(* IEC 61131-3 sources: RL_MAR/experiments/comparison/autoplc/results/gpt-4o-mini_20260511_164212/med_70, 1 file *)

(* ---- med_70_1.st ---- *)
FUNCTION_BLOCK EggIncubatorControl
    VAR_INPUT
        StartButton : BOOL; (* Input for starting the incubation process *)
        StopButton : BOOL; (* Input for stopping the incubation process *)
        TemperatureSensor : REAL; (* Input for temperature reading in °C *)
        HumiditySensor : REAL; (* Input for humidity reading in % *)
    END_VAR

    VAR_OUTPUT
        HeatingElement : BOOL; (* Output for controlling the heating element *)
        Humidifier : BOOL; (* Output for controlling the humidifier *)
        EggTurningMotor : BOOL; (* Output for controlling the egg turning motor *)
        IncubationInProgress : BOOL; (* Indicator for an ongoing incubation process *)
    END_VAR

    VAR
        TargetTemperature : REAL; (* Target temperature in °C *)
        TargetHumidity : REAL; (* Target humidity in % *)
        TurnIntervalSeconds : INT; (* Interval for turning eggs (1 hour in seconds) *)
        TurnTimerSeconds : INT; (* Timer for egg turning cycle in seconds *)
    END_VAR

    // Initialize control parameters
    TargetTemperature := 37.5;
    TargetHumidity := 50.0;
    TurnIntervalSeconds := 3600;
    TurnTimerSeconds := 0;

    // Main control logic
    IF StartButton AND NOT IncubationInProgress THEN
        IncubationInProgress := TRUE; // Start incubation
    END_IF;

    IF StopButton THEN
        IncubationInProgress := FALSE; // Stop incubation
        HeatingElement := FALSE; // Turn off heating element
        Humidifier := FALSE; // Turn off humidifier
        EggTurningMotor := FALSE; // Turn off egg turning motor
        TurnTimerSeconds := 0; // Reset timer
    END_IF;

    // Temperature control logic
    IF TemperatureSensor < TargetTemperature THEN
        HeatingElement := TRUE; // Turn on heating element
    ELSE
        HeatingElement := FALSE; // Turn off heating element
    END_IF;

    // Humidity control logic
    IF HumiditySensor < TargetHumidity THEN
        Humidifier := TRUE; // Turn on humidifier
    ELSE
        Humidifier := FALSE; // Turn off humidifier
    END_IF;

    // Egg turning cycle logic
    IF IncubationInProgress THEN
        TurnTimerSeconds := TurnTimerSeconds + 1; // Increment timer (assume this block is called every second)

        IF TurnTimerSeconds >= TurnIntervalSeconds THEN
            EggTurningMotor := NOT EggTurningMotor; // Toggle egg turning motor state
            TurnTimerSeconds := 0; // Reset timer
        END_IF;
    END_IF;

    // Update incubation status
    IncubationInProgress := IncubationInProgress; // This line is redundant but included for clarity
END_FUNCTION_BLOCK
